FUNCTION_BLOCK PUBLIC FB_Subscriber IMPLEMENTS I_Subscriber
VAR
	_Value				: LREAL;
END_VAR

PROPERTY ActualValue : LREAL
GET
ActualValue := THIS^._Value;
END_GET
END_PROPERTY

METHOD PUBLIC Update : BOOL
VAR_INPUT
	Value	: LREAL;
END_VAR
THIS^._Value := Value;
END_METHOD

END_FUNCTION_BLOCK

(* stored: Version 1.1.0.1, ProductVersion 3.1.4022.18
   POU FB_Subscriber: Id {40122c7b-204f-4d8a-8934-d01a04594cc3}, SpecialFunc None
   Property ActualValue: Id {bfb72149-d202-4acb-8317-036f3b16962d}
   Get Get: Id {a97714f2-db45-4076-9b3d-9c5a1c6910e5}
   Method Update: Id {ab10fc4b-83d9-407a-af6c-0bdbb13792fb} *)
